// TIA Portal V17 export
// export: Created 2024-09-02T12:50:05.0707784Z, ExportSetting WithDefaults, DisplayName Totally Integrated Automation Portal, DisplayVersion V17, DisplayName TIA Portal Openness, DisplayVersion V17, DisplayName TIA Portal Version Control Interface, DisplayVersion V17, DisplayName STEP 7 Professional, DisplayVersion V17, DisplayName STEP 7 Safety, DisplayVersion V17, DisplayName WinCC Professional, DisplayVersion V17
FUNCTION_BLOCK "FB190_Omron_Comunication"   // FB180, LAD
{ S7_Optimized_Access := 'FALSE' }
VERSION : 0.1
// stored: AutoNumber false, IsIECCheckEnabled false, SetENOAutomatically false, UDAEnableTagReadback false
   VAR_INPUT
      IO_Adress : Int;
      iRange_Input : Int;
      iRange_Output : Int;
      iProgram_Nr : Int;
      iExe_or_Step : Bool;
      i_Trigger : Bool;
      i_ReadTimeout : Time;
      i_ResetStatus : Bool;
      i_Ack : Bool;
   END_VAR
   VAR_OUTPUT
      q_Ready : Bool;
      q_Busy : Bool;
      q_Done : Bool;
      q_OK : Bool;
      q_NOK : Bool;
      q_Error : Bool;
      q_ErrorCode : Int;
      q_Data : Array[0..7] of DWord;
   END_VAR
   VAR DB_SPECIFIC
      Reserve : Array[0..11] of Byte;
      Interface : Struct
         PLC_Input : Struct
            Control_Input : Struct
               Reserve_3_0 : Bool;
               Reserve_3_1 : Bool;
               Reserve_3_2 : Bool;
               Reserve_3_3 : Bool;
               Reserve_3_4 : Bool;
               Reserve_3_5 : Bool;
               Reserve_3_6 : Bool;
               Reserve_3_7 : Bool;
               Gate : Bool;
               Reserve_2_1 : Bool;
               Reserve_2_2 : Bool;
               Reserve_2_3 : Bool;
               Reserve_2_4 : Bool;
               Reserve_2_5 : Bool;
               Reserve_2_6 : Bool;
               Reserve_2_7 : Bool;
               XFlag : Bool;
               Xbusy : Bool;
               xWait : Bool;
               Reserve_1_3 : Bool;
               Reserve_1_4 : Bool;
               Reserve_1_5 : Bool;
               Reserve_1_6 : Bool;
               Err : Bool;
               Flg : Bool;
               Busy : Bool;
               Reserve_0_2 : Bool;
               "OR" : Bool;
               Run : Bool;
               Ack : Bool;
               Reserve_0_6 : Bool;
               Reserve_0_7 : Bool;
            END_STRUCT;
            "CMD-CODE_2" : Word;
            "CMD-CODE_3" : Word;
            "RES-CODE" : DWord;
            "RES-DATA" : DWord;
            DATA0 : DWord;
            DATA1 : DWord;
            DATA2 : DWord;
            DATA3 : DWord;
            DATA4 : DWord;
            DATA5 : DWord;
            DATA6 : DWord;
            DATA7 : DWord;
            UserOutputArea0 : DWord;
            UserOutputArea1 : DWord;
            UserOutputArea2 : DWord;
            UserOutputArea3 : DWord;
            UserOutputArea4 : DWord;
            UserOutputArea5 : DWord;
         END_STRUCT;
         PLC_Output : Struct
            Control_Output : Struct
               Reserve_3_0 : Bool;
               Reserve_3_1 : Bool;
               Reserve_3_2 : Bool;
               Reserve_3_3 : Bool;
               Reserve_3_4 : Bool;
               Reserve_3_5 : Bool;
               Reserve_3_6 : Bool;
               Reserve_3_7 : Bool;
               Das : Bool;
               Reserve_2_1 : Bool;
               Reserve_2_2 : Bool;
               Reserve_2_3 : Bool;
               Reserve_2_4 : Bool;
               Reserve_2_5 : Bool;
               Reserve_2_6 : Bool;
               Reserve_2_7 : Bool;
               XExe : Bool;
               Reserve_1_1 : Bool;
               Reserve_1_2 : Bool;
               Reserve_1_3 : Bool;
               Reserve_1_4 : Bool;
               Reserve_1_5 : Bool;
               Reserve_1_6 : Bool;
               ErCLR : Bool;
               Exe : Bool;
               "Step" : Bool;
               Reserve_0_2 : Bool;
               Reserve_0_3 : Bool;
               Reserve_0_4 : Bool;
               Reserve_0_5 : Bool;
               Reserve_0_6 : Bool;
               Reserve_0_7 : Bool;
            END_STRUCT;
            "CMD-CODE_3" : Word;
            "CMD-CODE_2" : Word;
            "CMD-PARAM_1_5" : Word;
            "CMD-PARAM_1_4" : Word;
            "CMD-PARAM_2_7" : Word;
            "CMD-PARAM_2_6" : Word;
            "CMD-PARAM_3_9" : Word;
            "CMD-PARAM_3_8" : Word;
            UserInputArea0_11 : Word;
            UserInputArea0_10 : Word;
            UserInputArea1_13 : Word;
            UserInputArea1_12 : Word;
            UserInputArea2_15 : Word;
            UserInputArea2_14 : Word;
            UserInputArea3_17 : Word;
            UserInputArea3_16 : Word;
            UserInputArea4_1_19 : Word;
            UserInputArea4_1_18 : Word;
            UserInputArea4_2_21 : Word;
            UserInputArea4_2_20 : Word;
            UserInputArea5_1_23 : Word;
            UserInputArea5_1_22 : Word;
            UserInputArea5_2_25 : Word;
            UserInputArea5_2_24 : Word;
         END_STRUCT;
      END_STRUCT;
      t_Clear { ExternalAccessible := 'False'; ExternalVisible := 'False'; ExternalWritable := 'False'} : Bool;
      sReadComplete : Bool;
      sTrigHelpEdge : Bool;
      sReadTimeout : Bool;
      sReadTimer { ExternalAccessible := 'False'; ExternalVisible := 'False'; ExternalWritable := 'False'; S7_SetPoint := 'True'} : Array[0..3] of IEC_TIMER;
      sP_Trig_OR { S7_SetPoint := 'True'} : Bool;
   END_VAR
   VAR_TEMP
      ret_val : Int;
      i : Int;
      j : Int;
      k_data : Int;
      l_data : Int;
      Empty_Value : Int;
      tSaveFirstWord : Word;
      tSaveSecondWord : Word;
      tSaveFirstWord_Read : Word;
      tSaveSecondWord_Read : Word;
      t_InterfacePLCInput : Array[0..143] of Byte;
      t_InterfacePLCOutput : Array[0..19] of Byte;
      t_CMD_OK : Bool;
      t_CMD_OK_Read : Bool;
      copy_Data : Bool;
      Always_False : Bool;
   END_VAR
   VAR_TEMP   // added for the SCL form of the ladder/FBD networks
      _w1 : Bool;
      _w2 : Bool;
   END_VAR
BEGIN

REGION Network 1: Init
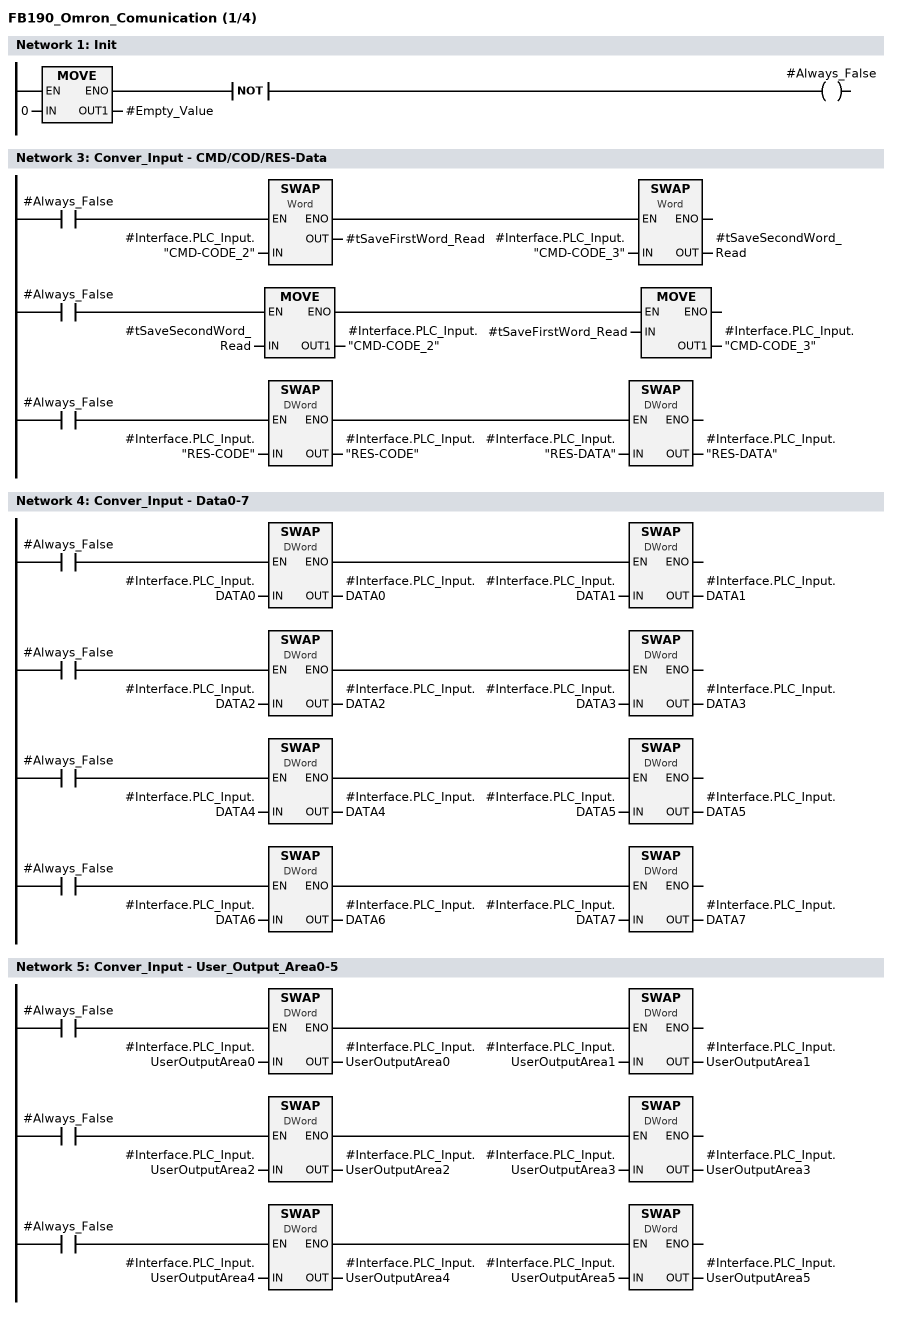
   RUNG wire#powerrail
      Move(in := 0, out1 => #Empty_Value)
      Not()
      Coil( #Always_False )
   END_RUNG
   // the same network as SCL:
   #Empty_Value := 0;
   #Always_False := NOT TRUE;
END_REGION

REGION Network 2 (SCL): Read Input PLC Area and copy to Stat
   FOR #i := 0 TO #iRange_Input BY 1
   DO
       #t_InterfacePLCInput [#i] := PEEK(area := 16#81,
                                       dbNumber := 0,
                                       byteOffset := #IO_Adress + #i);
   END_FOR;

   #ret_val := BLKMOV(SRCBLK := #t_InterfacePLCInput, DSTBLK => #Interface.PLC_Input);
END_REGION

REGION Network 3: Conver_Input - CMD/COD/RES-Data
   IF #Always_False THEN
       #tSaveFirstWord_Read := SWAP(#Interface.PLC_Input."CMD-CODE_2");
       #tSaveSecondWord_Read := SWAP(#Interface.PLC_Input."CMD-CODE_3");
       #Interface.PLC_Input."CMD-CODE_2" := #tSaveSecondWord_Read;
       #Interface.PLC_Input."CMD-CODE_3" := #tSaveFirstWord_Read;
       #Interface.PLC_Input."RES-CODE" := SWAP(#Interface.PLC_Input."RES-CODE");
       #Interface.PLC_Input."RES-DATA" := SWAP(#Interface.PLC_Input."RES-DATA");
   END_IF;
END_REGION

REGION Network 4: Conver_Input - Data0-7
   IF #Always_False THEN
       #Interface.PLC_Input.DATA0 := SWAP(#Interface.PLC_Input.DATA0);
       #Interface.PLC_Input.DATA1 := SWAP(#Interface.PLC_Input.DATA1);
       #Interface.PLC_Input.DATA2 := SWAP(#Interface.PLC_Input.DATA2);
       #Interface.PLC_Input.DATA3 := SWAP(#Interface.PLC_Input.DATA3);
       #Interface.PLC_Input.DATA4 := SWAP(#Interface.PLC_Input.DATA4);
       #Interface.PLC_Input.DATA5 := SWAP(#Interface.PLC_Input.DATA5);
       #Interface.PLC_Input.DATA6 := SWAP(#Interface.PLC_Input.DATA6);
       #Interface.PLC_Input.DATA7 := SWAP(#Interface.PLC_Input.DATA7);
   END_IF;
END_REGION

REGION Network 5: Conver_Input - User_Output_Area0-5
   IF #Always_False THEN
       #Interface.PLC_Input.UserOutputArea0 := SWAP(#Interface.PLC_Input.UserOutputArea0);
       #Interface.PLC_Input.UserOutputArea1 := SWAP(#Interface.PLC_Input.UserOutputArea1);
       #Interface.PLC_Input.UserOutputArea2 := SWAP(#Interface.PLC_Input.UserOutputArea2);
       #Interface.PLC_Input.UserOutputArea3 := SWAP(#Interface.PLC_Input.UserOutputArea3);
       #Interface.PLC_Input.UserOutputArea4 := SWAP(#Interface.PLC_Input.UserOutputArea4);
       #Interface.PLC_Input.UserOutputArea5 := SWAP(#Interface.PLC_Input.UserOutputArea5);
   END_IF;
END_REGION

REGION Network 6: ##########################
END_REGION

REGION Network 7: Ready status
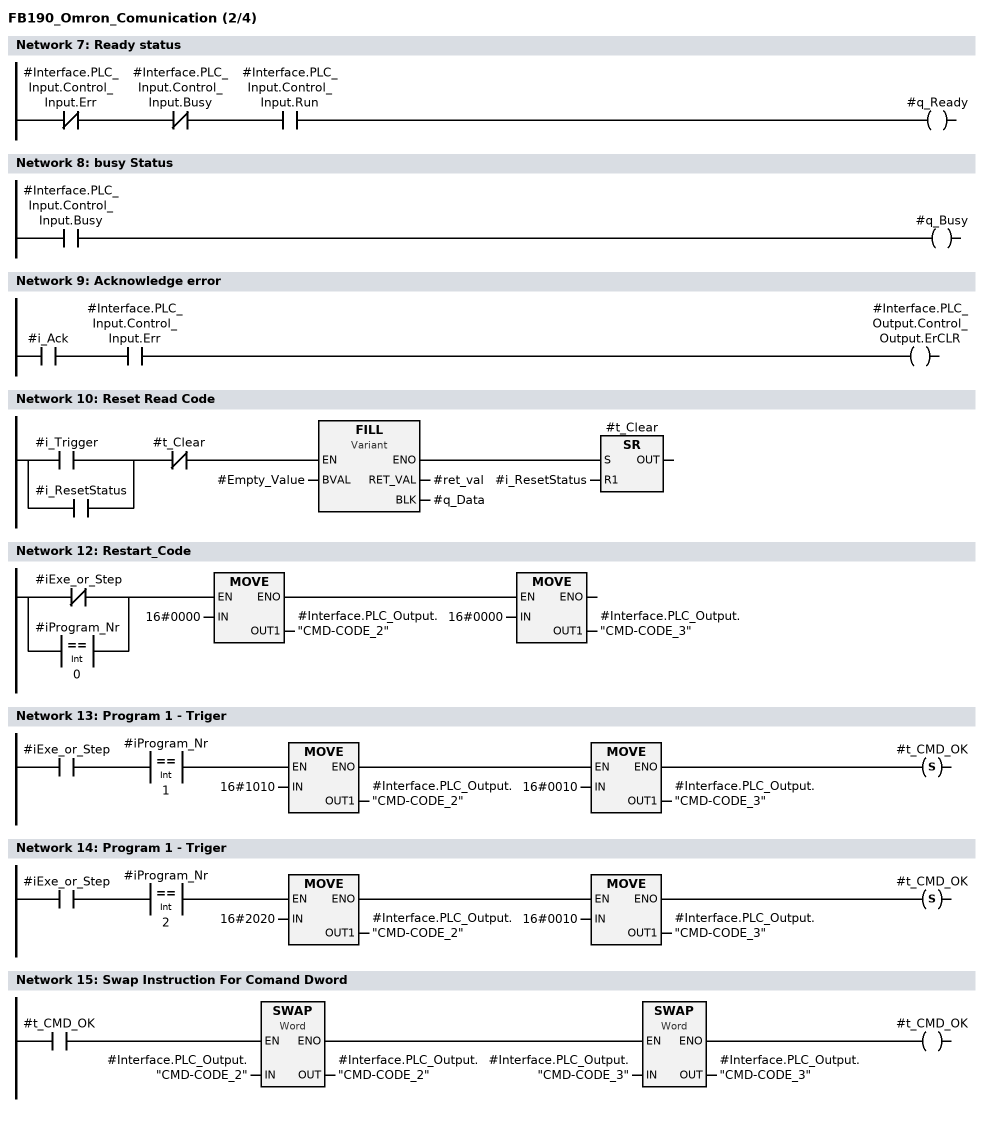
   RUNG wire#powerrail
      I_Contact( #Interface.PLC_Input.Control_Input.Err )
      I_Contact( #Interface.PLC_Input.Control_Input.Busy )
      Contact( #Interface.PLC_Input.Control_Input.Run )
      Coil( #q_Ready )
   END_RUNG
   // the same network as SCL:
   #q_Ready := NOT #Interface.PLC_Input.Control_Input.Err AND NOT #Interface.PLC_Input.Control_Input.Busy AND #Interface.PLC_Input.Control_Input.Run;
END_REGION

REGION Network 8: busy Status
   RUNG wire#powerrail
      Contact( #Interface.PLC_Input.Control_Input.Busy )
      Coil( #q_Busy )
   END_RUNG
   // the same network as SCL:
   #q_Busy := #Interface.PLC_Input.Control_Input.Busy;
END_REGION

REGION Network 9: Acknowledge error
   RUNG wire#powerrail
      Contact( #i_Ack )
      Contact( #Interface.PLC_Input.Control_Input.Err )
      Coil( #Interface.PLC_Output.Control_Output.ErCLR )
   END_RUNG
   // the same network as SCL:
   #Interface.PLC_Output.Control_Output.ErCLR := #i_Ack AND #Interface.PLC_Input.Control_Input.Err;
END_REGION

REGION Network 10: Reset Read Code
   RUNG wire#powerrail
      Contact( #i_Trigger )
      wire#w1
      I_Contact( #t_Clear )
      { S7_Templates := "ptr_type := Variant" } FILL(BVAL := #Empty_Value, RET_VAL => #ret_val, BLK => #q_Data)
      S_SR(operand := #t_Clear, r1 := #i_ResetStatus)
   END_RUNG
   RUNG wire#powerrail
      Contact( #i_ResetStatus )
   END_RUNG wire#w1
   // the same network as SCL:
   #_w1 := (#i_Trigger OR #i_ResetStatus) AND NOT #t_Clear;
   #ret_val := FILL(EN := #_w1, BVAL := #Empty_Value, BLK => #q_Data, ENO => #_w2);
   IF #_w2 THEN
       #t_Clear := TRUE;   // SR flip-flop
   END_IF;
   IF #i_ResetStatus THEN #t_Clear := FALSE; END_IF;
END_REGION

REGION Network 11: #######Load Commend#######
END_REGION

REGION Network 12: Restart_Code
   RUNG wire#powerrail
      I_Contact( #iExe_or_Step )
      wire#w1
      Move(in := 16#0000, out1 => #Interface.PLC_Output."CMD-CODE_2")
      Move(in := 16#0000, out1 => #Interface.PLC_Output."CMD-CODE_3")
   END_RUNG
   RUNG wire#powerrail
      { S7_Templates := "SrcType := Int" } EQ_Contact(in1 := #iProgram_Nr, in2 := 0)
   END_RUNG wire#w1
   // the same network as SCL:
   IF NOT #iExe_or_Step OR (#iProgram_Nr = 0) THEN
       #Interface.PLC_Output."CMD-CODE_2" := 16#0000;
       #Interface.PLC_Output."CMD-CODE_3" := 16#0000;
   END_IF;
END_REGION

REGION Network 13: Program 1 - Triger
   RUNG wire#powerrail
      Contact( #iExe_or_Step )
      { S7_Templates := "SrcType := Int" } EQ_Contact(in1 := #iProgram_Nr, in2 := 1)
      Move(in := 16#1010, out1 => #Interface.PLC_Output."CMD-CODE_2")
      Move(in := 16#0010, out1 => #Interface.PLC_Output."CMD-CODE_3")
      S_Coil( #t_CMD_OK )
   END_RUNG
   // the same network as SCL:
   IF #iExe_or_Step AND (#iProgram_Nr = 1) THEN
       #Interface.PLC_Output."CMD-CODE_2" := 16#1010;
       #Interface.PLC_Output."CMD-CODE_3" := 16#0010;
       #t_CMD_OK := TRUE;
   END_IF;
END_REGION

REGION Network 14: Program 1 - Triger
   RUNG wire#powerrail
      Contact( #iExe_or_Step )
      { S7_Templates := "SrcType := Int" } EQ_Contact(in1 := #iProgram_Nr, in2 := 2)
      Move(in := 16#2020, out1 => #Interface.PLC_Output."CMD-CODE_2")
      Move(in := 16#0010, out1 => #Interface.PLC_Output."CMD-CODE_3")
      S_Coil( #t_CMD_OK )
   END_RUNG
   // the same network as SCL:
   IF #iExe_or_Step AND (#iProgram_Nr = 2) THEN
       #Interface.PLC_Output."CMD-CODE_2" := 16#2020;
       #Interface.PLC_Output."CMD-CODE_3" := 16#0010;
       #t_CMD_OK := TRUE;
   END_IF;
END_REGION

REGION Network 15: Swap Instruction For Comand Dword
   IF #t_CMD_OK THEN
       #Interface.PLC_Output."CMD-CODE_2" := SWAP(#Interface.PLC_Output."CMD-CODE_2");
       #Interface.PLC_Output."CMD-CODE_3" := SWAP(#Interface.PLC_Output."CMD-CODE_3");
   END_IF;
   #t_CMD_OK := #t_CMD_OK;
END_REGION

REGION Network 16: -----------------------------------------------------------------
END_REGION

REGION Network 17: Request Start Reading
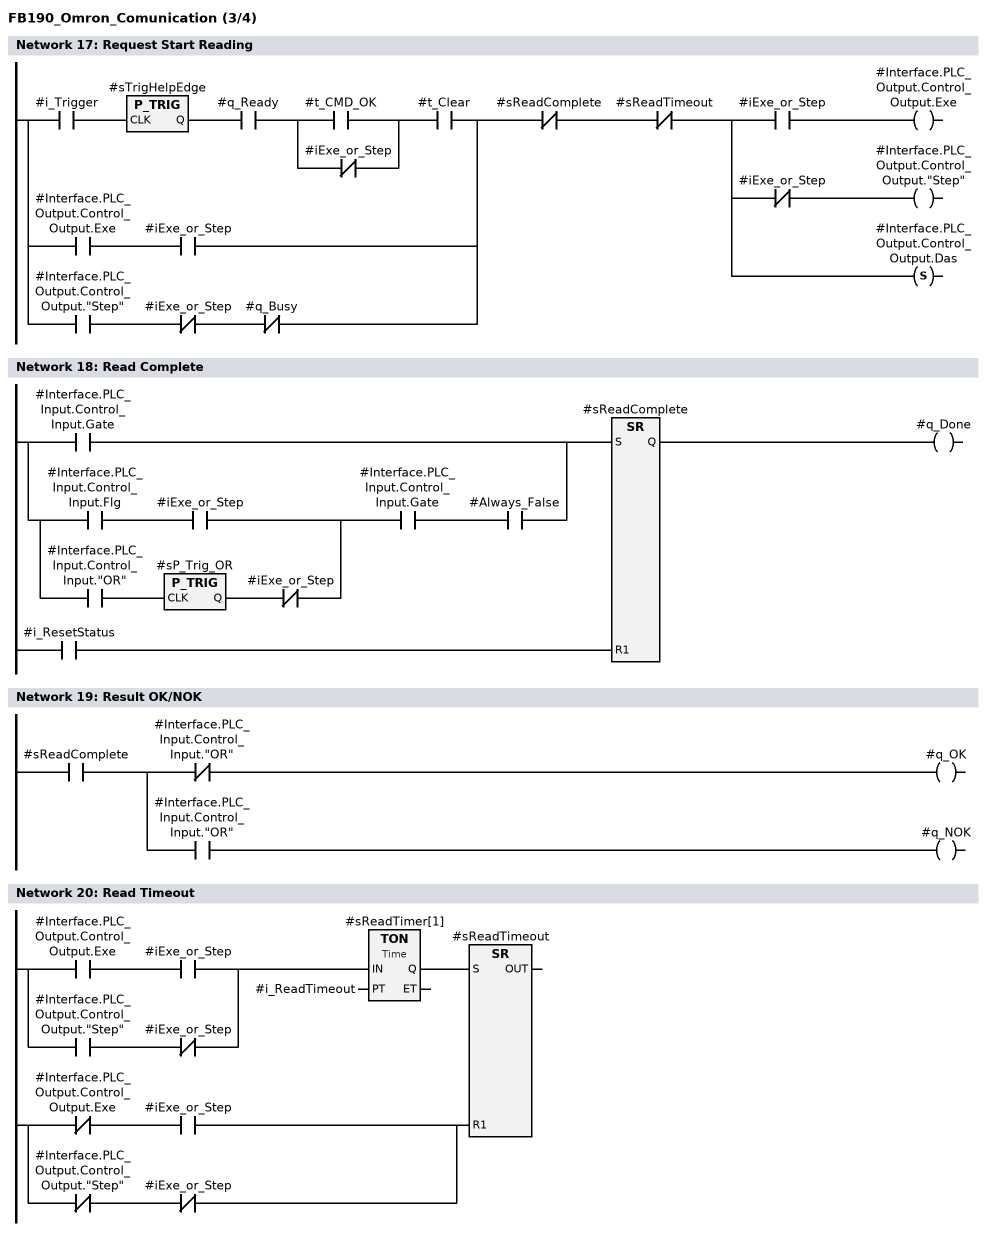
   RUNG wire#powerrail
      Contact( #i_Trigger )
      P_Trig( #sTrigHelpEdge )
      Contact( #q_Ready )
      wire#w1
      Contact( #t_CMD_OK )
      wire#w2
      Contact( #t_Clear )
      wire#w3
      I_Contact( #sReadComplete )
      I_Contact( #sReadTimeout )
      wire#w4
      Contact( #iExe_or_Step )
      Coil( #Interface.PLC_Output.Control_Output.Exe )
   END_RUNG
   RUNG wire#w1
      I_Contact( #iExe_or_Step )
   END_RUNG wire#w2
   RUNG wire#powerrail
      Contact( #Interface.PLC_Output.Control_Output.Exe )
      Contact( #iExe_or_Step )
   END_RUNG wire#w3
   RUNG wire#powerrail
      Contact( #Interface.PLC_Output.Control_Output."Step" )
      I_Contact( #iExe_or_Step )
      I_Contact( #q_Busy )
   END_RUNG wire#w3
   RUNG wire#w4
      I_Contact( #iExe_or_Step )
      Coil( #Interface.PLC_Output.Control_Output."Step" )
   END_RUNG
   RUNG wire#w4
      S_Coil( #Interface.PLC_Output.Control_Output.Das )
   END_RUNG
   // the same network as SCL:
   #_w1 := #i_Trigger AND NOT #sTrigHelpEdge;   // rising edge
   #sTrigHelpEdge := #i_Trigger;
   #_w2 := ((#_w1 AND #q_Ready AND (#t_CMD_OK OR NOT #iExe_or_Step) AND #t_Clear) OR (#Interface.PLC_Output.Control_Output.Exe AND #iExe_or_Step) OR (#Interface.PLC_Output.Control_Output."Step" AND NOT #iExe_or_Step AND NOT #q_Busy)) AND NOT #sReadComplete AND NOT #sReadTimeout;
   #Interface.PLC_Output.Control_Output.Exe := #_w2 AND #iExe_or_Step;
   #Interface.PLC_Output.Control_Output."Step" := #_w2 AND NOT #iExe_or_Step;
   IF #_w2 THEN #Interface.PLC_Output.Control_Output.Das := TRUE; END_IF;
END_REGION

REGION Network 18: Read Complete
   RUNG wire#powerrail
      Contact( #Interface.PLC_Input.Control_Input.Gate )
      wire#w1
      S_SR(operand := #sReadComplete, r1 := wire#w3)
      Coil( #q_Done )
   END_RUNG
   RUNG wire#powerrail
      Contact( #Interface.PLC_Input.Control_Input.Flg )
      Contact( #iExe_or_Step )
      wire#w2
      Contact( #Interface.PLC_Input.Control_Input.Gate )
      Contact( #Always_False )
   END_RUNG wire#w1
   RUNG wire#powerrail
      Contact( #Interface.PLC_Input.Control_Input."OR" )
      P_Trig( #sP_Trig_OR )
      I_Contact( #iExe_or_Step )
   END_RUNG wire#w2
   RUNG wire#powerrail
      Contact( #i_ResetStatus )
   END_RUNG wire#w3
   // the same network as SCL:
   #_w1 := #Interface.PLC_Input.Control_Input."OR" AND NOT #sP_Trig_OR;   // rising edge
   #sP_Trig_OR := #Interface.PLC_Input.Control_Input."OR";
   IF #Interface.PLC_Input.Control_Input.Gate OR (((#Interface.PLC_Input.Control_Input.Flg AND #iExe_or_Step) OR (#_w1 AND NOT #iExe_or_Step)) AND #Interface.PLC_Input.Control_Input.Gate AND #Always_False) THEN
       #sReadComplete := TRUE;   // SR flip-flop
   END_IF;
   IF #i_ResetStatus THEN #sReadComplete := FALSE; END_IF;
   #q_Done := #sReadComplete;
END_REGION

REGION Network 19: Result OK/NOK
   RUNG wire#powerrail
      Contact( #sReadComplete )
      wire#w1
      I_Contact( #Interface.PLC_Input.Control_Input."OR" )
      Coil( #q_OK )
   END_RUNG
   RUNG wire#w1
      Contact( #Interface.PLC_Input.Control_Input."OR" )
      Coil( #q_NOK )
   END_RUNG
   // the same network as SCL:
   #q_OK := #sReadComplete AND NOT #Interface.PLC_Input.Control_Input."OR";
   #q_NOK := #sReadComplete AND #Interface.PLC_Input.Control_Input."OR";
END_REGION

REGION Network 20: Read Timeout
   RUNG wire#powerrail
      Contact( #Interface.PLC_Output.Control_Output.Exe )
      Contact( #iExe_or_Step )
      wire#w1
      { S7_Templates := "time_type := Time" } #sReadTimer[1].TON(pt := #i_ReadTimeout, et =>)
      S_SR(operand := #sReadTimeout, r1 := wire#w2)
   END_RUNG
   RUNG wire#powerrail
      Contact( #Interface.PLC_Output.Control_Output."Step" )
      I_Contact( #iExe_or_Step )
   END_RUNG wire#w1
   RUNG wire#powerrail
      I_Contact( #Interface.PLC_Output.Control_Output.Exe )
      Contact( #iExe_or_Step )
   END_RUNG wire#w2
   RUNG wire#powerrail
      I_Contact( #Interface.PLC_Output.Control_Output."Step" )
      I_Contact( #iExe_or_Step )
   END_RUNG wire#w2
   // the same network as SCL:
   #sReadTimer[1].TON(IN := (#Interface.PLC_Output.Control_Output.Exe AND #iExe_or_Step) OR (#Interface.PLC_Output.Control_Output."Step" AND NOT #iExe_or_Step),
                      PT := #i_ReadTimeout);
   IF #sReadTimer[1].Q THEN
       #sReadTimeout := TRUE;   // SR flip-flop
   END_IF;
   IF (NOT #Interface.PLC_Output.Control_Output.Exe AND #iExe_or_Step) OR (NOT #Interface.PLC_Output.Control_Output."Step" AND NOT #iExe_or_Step) THEN
       #sReadTimeout := FALSE;
   END_IF;
END_REGION

REGION Network 21: Copy Data
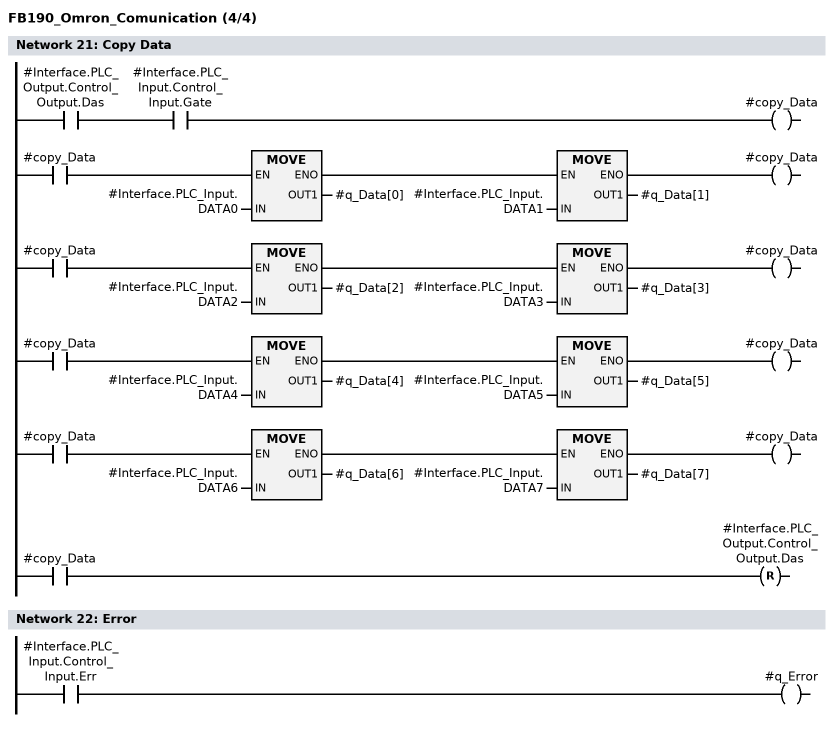
   RUNG wire#powerrail
      Contact( #Interface.PLC_Output.Control_Output.Das )
      Contact( #Interface.PLC_Input.Control_Input.Gate )
      Coil( #copy_Data )
   END_RUNG
   RUNG wire#powerrail
      Contact( #copy_Data )
      Move(in := #Interface.PLC_Input.DATA0, out1 => #q_Data[0])
      Move(in := #Interface.PLC_Input.DATA1, out1 => #q_Data[1])
      Coil( #copy_Data )
   END_RUNG
   RUNG wire#powerrail
      Contact( #copy_Data )
      Move(in := #Interface.PLC_Input.DATA2, out1 => #q_Data[2])
      Move(in := #Interface.PLC_Input.DATA3, out1 => #q_Data[3])
      Coil( #copy_Data )
   END_RUNG
   RUNG wire#powerrail
      Contact( #copy_Data )
      Move(in := #Interface.PLC_Input.DATA4, out1 => #q_Data[4])
      Move(in := #Interface.PLC_Input.DATA5, out1 => #q_Data[5])
      Coil( #copy_Data )
   END_RUNG
   RUNG wire#powerrail
      Contact( #copy_Data )
      Move(in := #Interface.PLC_Input.DATA6, out1 => #q_Data[6])
      Move(in := #Interface.PLC_Input.DATA7, out1 => #q_Data[7])
      Coil( #copy_Data )
   END_RUNG
   RUNG wire#powerrail
      Contact( #copy_Data )
      R_Coil( #Interface.PLC_Output.Control_Output.Das )
   END_RUNG
   // the same network as SCL:
   #copy_Data := #Interface.PLC_Output.Control_Output.Das AND #Interface.PLC_Input.Control_Input.Gate;
   IF #copy_Data THEN
       #q_Data[0] := #Interface.PLC_Input.DATA0;
       #q_Data[1] := #Interface.PLC_Input.DATA1;
   END_IF;
   #copy_Data := #copy_Data;
   IF #copy_Data THEN
       #q_Data[2] := #Interface.PLC_Input.DATA2;
       #q_Data[3] := #Interface.PLC_Input.DATA3;
   END_IF;
   #copy_Data := #copy_Data;
   IF #copy_Data THEN
       #q_Data[4] := #Interface.PLC_Input.DATA4;
       #q_Data[5] := #Interface.PLC_Input.DATA5;
   END_IF;
   #copy_Data := #copy_Data;
   IF #copy_Data THEN
       #q_Data[6] := #Interface.PLC_Input.DATA6;
       #q_Data[7] := #Interface.PLC_Input.DATA7;
   END_IF;
   #copy_Data := #copy_Data;
   IF #copy_Data THEN #Interface.PLC_Output.Control_Output.Das := FALSE; END_IF;
END_REGION

REGION Network 22: Error
   RUNG wire#powerrail
      Contact( #Interface.PLC_Input.Control_Input.Err )
      Coil( #q_Error )
   END_RUNG
   // the same network as SCL:
   #q_Error := #Interface.PLC_Input.Control_Input.Err;
END_REGION

REGION Network 23 (SCL): Write Output PLC Area
   #ret_val := BLKMOV(SRCBLK := #Interface.PLC_Output, DSTBLK => #t_InterfacePLCOutput);

   FOR #j := 0 TO #iRange_Output BY 1 DO
       POKE(area := 16#82,
            dbNumber := 0,
            byteOffset := #IO_Adress  + #j,
            value := #t_InterfacePLCOutput[#j]);
   END_FOR;
END_REGION
END_FUNCTION_BLOCK
